// TwinCAT 3 PLC project CleanroomConnect
// ProgramVersion: 3.1.4024.0
// libraries:
//   KMWE Generic Library, * (KMWE)
//   Tc2_MC2, * (Beckhoff Automation GmbH)
//   Tc2_Standard, * (Beckhoff Automation GmbH)
//   Tc2_System, * (Beckhoff Automation GmbH)
//   Tc2_Utilities, * (Beckhoff Automation GmbH)
//   Tc3_Module, * (Beckhoff Automation GmbH)
//   VisuDialogs, * (System)
//   VisuSymbols,3.5.10.0,System
// project tree:
//   DUTs/ E_CtrlState.TcDUT (not stored), I_Door.TcIO (not stored), I_Servo.TcIO, ST_HmiBottomBar.TcDUT, ST_HmiMiddle.TcDUT, ST_HmiTopBar.TcDUT
//   / GlobalTextList.TcGTLO, MAIN.TcPOU, PlcTask.TcTTO (not stored)
//   GVLs/ GVL.TcGVL, GVL_Modules.TcGVL
//   POUs/02 UN/Unit %28UN%29/DUT/ E_AirState.TcDUT (not stored), E_ReqAction.TcDUT (not stored), E_SeqCleanroomConnect.TcDUT (not stored), ST_UN_CleanroomConnectSettings.TcDUT (not stored)
//   POUs/02 UN/Unit %28UN%29/ UN_CleanroomConnect.TcPOU (not stored)
//   POUs/03 EM/Equipment %28EM%29/2 EM_PalletConveyor/DUT/ E_ActionSelection.TcDUT (not stored), E_SeqPalletConveyor.TcDUT (not stored), I_EM_PalletConveyor.TcIO (not stored), ST_SettingsPalletConveyor.TcDUT (not stored)
//   POUs/03 EM/Equipment %28EM%29/3 EM_DockingInterface/DUTs/ I_EM_DockingInterface.TcIO (not stored), E_SeqDockingInterface.TcDUT (not stored), ST_SettingsDockingInterface.TcDUT (not stored)
//   POUs/03 EM/Equipment %28EM%29/4 EM_LiftingTransport/DUT/ E_SeqLiftingTransport.TcDUT (not stored), I_EM_LiftingTransport.TcIO (not stored), ST_PositioningProfile.TcDUT (not stored), ST_SettingsLiftingTransport.TcDUT (not stored)
//   POUs/03 EM/Equipment %28EM%29/EM_AirTreatment/DUTs/ E_SeqAirTreatment.TcDUT (not stored), I_EM_AirTreatment.TcIO (not stored), ST_SettingsAirTreatment.TcDUT (not stored)
//   POUs/03 EM/Equipment %28EM%29/EM_AirTreatment/ EM_AirTreatment.TcPOU (not stored)
//   POUs/03 EM/Equipment %28EM%29/4 EM_LiftingTransport/ EM_LiftingTransport.TcPOU (not stored)
//   POUs/03 EM/Equipment %28EM%29/1 EM_Utilities/DUTs/ E_ForceValue.TcDUT (not stored), I_EM_Utilities.TcIO (not stored), ST_SettingsUtilities.TcDUT (not stored)
//   POUs/03 EM/Equipment %28EM%29/1 EM_Utilities/ EM_Utilities.TcPOU (not stored)
//   POUs/03 EM/Equipment %28EM%29/3 EM_DockingInterface/ EM_DockingInterface.TcPOU (not stored)
//   POUs/03 EM/Equipment %28EM%29/2 EM_PalletConveyor/ EM_PalletConveyor.TcPOU (not stored)
//   POUs/04 CM/Control %28CM%29/CM_DIgitalOutput/DUT/ ST_DigOutput_HMI.TcDUT (not stored)
//   POUs/04 CM/Control %28CM%29/CM_DoorLock/DUT/ E_SeqDoorLock.TcDUT (not stored), ST_DoorLock_HMI.TcDUT (not stored), ST_SettingsDoorLock.TcDUT (not stored)
//   POUs/04 CM/Control %28CM%29/CM_MoviTrac_B/DUT/ E_SeqMoviTrac_B_WithBrake.TcDUT (not stored), I_MoviTrac_B.TcIO (not stored), ST_MoviTrac_B_HMI.TcDUT (not stored), ST_SettingsMoviTrac_B_WithBrake.TcDUT (not stored)
//   POUs/04 CM/Control %28CM%29/CM_Servo/ CM_Servo.TcPOU (not stored)
//   POUs/04 CM/Control %28CM%29/CM_Servo/DUT/ E_SeqServo.TcDUT (not stored), E_SeqInit.TcDUT (not stored), I_ServoMotor.TcIO (not stored), ST_Servo_HMI.TcDUT (not stored), ST_SettingsServo.TcDUT (not stored)
//   POUs/04 CM/Control %28CM%29/CM_DIgitalOutput/ CM_DigOutput.TcPOU (not stored)
//   POUs/04 CM/Control %28CM%29/CM_MoviTrac_B/ CM_MoviTrac_B.TcPOU (not stored)
//   POUs/04 CM/Control %28CM%29/CM_SpeedDoor/DUT/ ST_SettingsSpeedDoor.TcDUT (not stored), ST_SpeedDoor_HMI.TcDUT (not stored)
//   POUs/04 CM/Control %28CM%29/CM_TubeLedRgb/ CM_TubeLedRgb.TcPOU (not stored)
//   POUs/04 CM/Control %28CM%29/CM_TubeLedRgb/DUT/ I_LedRgb.TcIO (not stored)
//   POUs/04 CM/Control %28CM%29/CM_SpeedDoor/ CM_SpeedDoor.TcPOU (not stored)
//   POUs/04 CM/Control %28CM%29/CM_DoorLock/ CM_DoorLock.TcPOU (not stored)
//   POUs/04 CM/Control %28CM%29/CM_ValveWithFB/ CM_ValveWithDoubleFB.TcPOU (not stored), CM_ValveWithFB.TcPOU (not stored)
//   POUs/04 CM/Control %28CM%29/CM_ValveWithFB/DUT/ ST_SettingsValveWithFB.TcDUT (not stored), ST_ValveWithFB_HMI.TcDUT (not stored)
//   POUs/General/ FB_Flash.TcPOU, FB_ForceOutput.TcPOU, FB_Interlock.TcPOU (not stored), FB_InterlockHandler.TcPOU, FB_ModeStateControl.TcPOU, FB_MovAvg.TcPOU, FB_Toggle.TcPOU, F_InRange.TcPOU, ST_Interlock.TcDUT, ST_InterlockList.TcDUT, ST_MsgBox.TcDUT
// real-time tasks:
//   TASK PlcTask: cycle T#10ms, priority 20, ADS port 350
//   TASK PlcTaskHwSim: cycle T#10ms, priority 21, ADS port 351
// motion (NC):
//   TASK NC-Task 1 SAF: cycle T#2ms, priority 4, ADS port 501
//   TASK NC-Task 1 SVB: cycle T#10ms, priority 8, ADS port 511
//   AXIS TransportUnit (id 2)
//     Dynamic: AccelerationMaximum=500, DecelerationMaximum=500, Acceleration=90.006, Deceleration=90.006, Jerk=270.018
//     Velo: RefSearch=0.60004, RefSync=0.60004, SlowManual=0.5, FastManual=5, Fast=60.004, Maximum=60.004
//     PositionAreaControl: Range=0.1
//     TargetPosControl: Range=0.1
//     OtherSettings: AllowMotionCmdToSlave=true
//     encoder EncType=19
//       EncPara: ScaleFactorNumerator=180.013259, ScaleFactorDenominator=52428800, Offset=5558.46862311247, MaxCount=#xffffffff, ReferenceSystem=3
//         SoftEndMinControl: Enable=true
//         SoftEndMaxControl: Enable=true, Range=870
//         Inc: RefSearchInverse=true, RefSyncInverse=false
//     drive DrvType=16
//       DrvPara: MaxCount=#xffffffff, DriveControlDWord=#x00020100
//         Analog: VeloReferenz=66.0044, VeloScale=32, TorqueSetpointScale=10, ScaleFactorActTorque=0.1
//         TimeComp: TaskDelayCycles=1
//     controller CtrType=1
//       CtrPara: PriorControlFactor=1
//         PosDiffControl: Range=0.02
//         Observer: BandWidth=20
//   AXIS ScissorLift (id 3)
//     Dynamic: AccelerationMaximum=5, DecelerationMaximum=5, Acceleration=5, Deceleration=5, Jerk=23.436
//     Velo: RefSearch=0.05208, RefSync=0.05208, SlowManual=0.25, FastManual=2.5, Fast=5.208, Maximum=5.208
//     PositionAreaControl: Range=0.1
//     TargetPosControl: Range=0.1
//     OtherSettings: AllowMotionCmdToSlave=true, PulseDistancePos=10, PulseDistanceNeg=10
//     encoder EncType=8
//       EncPara: ScaleFactorNumerator=6, ScaleFactorDenominator=50331648, Offset=46.5910750851166, MaxCount=#xffffffff, ReferenceSystem=3
//         SoftEndMinControl: Enable=true
//         SoftEndMaxControl: Enable=true, Range=152
//         Inc: RefSearchInverse=true, RefSyncInverse=false
//     drive DrvType=9
//       DrvPara: MaxCount=#xffffffff, DriveControlDWord=#x00030100
//         Analog: VeloReferenz=5.7288, VeloScale=1.02400649589962, TorqueSetpointScale=10, ScaleFactorActTorque=0.1
//         TimeComp: TaskDelayCycles=1
//     controller CtrType=1
//       CtrPara: PriorControlFactor=1
//         PosDiffControl: Range=0.01
//         Observer: BandWidth=20
// I/O:
//   DEVICE Master (EtherCAT), AmsNetId 5.152.40.20.4.1
//     K1 (EK1200) [EK1200-5000 EtherCAT Power supply (2A E-Bus)]
//       K2 (EL6070-0033) [EL6070-0033 1Ch. Licence key terminal, individual licences]
//       K3 (EL1809) [EL1809 16Ch. Dig. Input 24V, 3ms]
//       K4 (EL1809) [EL1809 16Ch. Dig. Input 24V, 3ms]
//       K5 (EL1809) [EL1809 16Ch. Dig. Input 24V, 3ms]
//       K6 (EL1809) [EL1809 16Ch. Dig. Input 24V, 3ms]
//       K7 (EL2809) [EL2809 16Ch. Dig. Output 24V, 0.5A]
//       K8 (EL4024) [EL4024 4Ch. Ana. Output 4-20mA, 12bit]
//       K9 (EL7211-9014) [EL7211-9014 1Ch. MDP742 Servo motor output stage with OCT (50V, 4.5A RMS) and STO input]
//         startup 32785:21 := 0E01 // DRV Motor Settings / Commutation offset
//         startup 32786:19 := 0000 // DRV Brake Settings / Emergency application timeout
//         startup 32784:51 := 0A00 // DRV Amplifier Settings / Stand still window
//         startup 32785:27 := 4F080000 // DRV Motor Settings / Motor speed limitation
//         startup 28688:3 := 09 // DRV Outputs / Modes of operation
//         startup 32784:87 := 64 // DRV Amplifier Settings / Velocity feed forward gain
//         startup 28688:11 := D007 // DRV Outputs / Torque limitation
//         startup 32784:19 := 8701 // DRV Amplifier Settings / Current loop proportional gain
//         startup 32784:18 := 0500 // DRV Amplifier Settings / Current loop integral time
//         startup 32784:21 := 92000000 // DRV Amplifier Settings / Velocity loop proportional gain
//         startup 32784:20 := 96000000 // DRV Amplifier Settings / Velocity loop integral time
//         startup 32768:1 := 00 // FB Settings / Invert feedback direction
//       K10 (EL9576) [EL9576 Brake chopper terminal]
//       K11 (EL2904) [EL2904, 4 Ch. Safety Output 24V, 0.5A, TwinSAFE]
//         modules: Module 1 (FSOES), Module 2 (DO)
//       K12 (EL1918 + TwinSAFE Logic)
//       K20 (EL9110) [EL9110 Power Supplier with LED (24V, Diagnostics)]
//       K21 (EL2809) [EL2809 16Ch. Dig. Output 24V, 0.5A]
//       K22 (EL9011) [EL9011 End Terminal]
//   DEVICE Master Field (EtherCAT), AmsNetId 5.152.40.20.5.1
//     U9 (AX5103-0000-0215) [AX5103-0000-0215 EtherCAT Drive (SoE, 1 Ch.)]
//       Term 3 (AX5805) [AX5805 (Safety Drive Option)]
//         modules: Module 1 (Safety Process Data, 1 axis), Module 2 (Standard Process Data, 1 axis)
//       Term 3 (EL9011) [EL9011 End Terminal]
// variable links:
//   Master (EtherCAT) <-> Master (EtherCAT)/K1 (EK1200)/K12 (EL1918 + TwinSAFE Logic)
//     K1 (EK1200)/K11 (EL2904)/Module 1 (FSOES)/RxPDO/FSOE <-> ConnectionInputs/TwinSafeGroup1.EL2904, 4 digital outputs_1_22 TxPDO
//     K1 (EK1200)/K11 (EL2904)/Module 1 (FSOES)/TxPDO/FSOE <-> ConnectionOutputs/TwinSafeGroup1.EL2904, 4 digital outputs_1_22 RxPDO
//   Master (EtherCAT) <-> Master Field (EtherCAT)/U9 (AX5103-0000-0215)/Term 3 (AX5805)
//     K1 (EK1200)/K12 (EL1918 + TwinSAFE Logic)/ConnectionInputs/TwinSafeGroup1.AX5805, Safety Process Data 1 axis_37 TxPDO <-> Module 1 (Safety Process Data, 1 axis)/Outputs (Controlword)/FSOE
//     K1 (EK1200)/K12 (EL1918 + TwinSAFE Logic)/ConnectionOutputs/TwinSafeGroup1.AX5805, Safety Process Data 1 axis_37 RxPDO <-> Module 1 (Safety Process Data, 1 axis)/Inputs (Statusword)/FSOE
//   NC-Task 1 SAF/Axes/TransportUnit <-> Master (EtherCAT)/K1 (EK1200)/K9 (EL7211-9014)
//     Drive/Inputs/In/nDataIn1 <-> DRV Following error actual value/Following error actual value
//     Drive/Inputs/In/nDataIn3[0] <-> DRV Torque actual value/Torque actual value
//     Drive/Inputs/In/nDcOutputTime <-> InfoData/DcOutputShift
//     Drive/Inputs/In/nState1 <-> DRV Statusword/Statusword
//     Drive/Inputs/In/nState2 <-> DRV Statusword/Statusword @bit 8
//     Drive/Inputs/In/nState4 @bit 1 <-> WcState/InputToggle
//     Drive/Inputs/In/nState4 <-> WcState/WcState
//     Drive/Outputs/Out/nCtrl1 <-> DRV Controlword/Controlword
//     Drive/Outputs/Out/nCtrl2 <-> DRV Controlword/Controlword @bit 8
//     Drive/Outputs/Out/nDataOut1 <-> DRV Target position/Target position
//     Drive/Outputs/Out/nDataOut2 <-> DRV Target velocity/Target velocity
//     Enc/Inputs/In/nDataIn1 <-> FB Position/Position
//     Enc/Inputs/In/nDcInputTime <-> InfoData/DcInputShift
//     Enc/Inputs/In/nState4 @bit 1 <-> WcState/InputToggle
//     Enc/Inputs/In/nState4 <-> WcState/WcState
//   CleanroomConnect/CleanroomConnect Instance <-> Master (EtherCAT)/K1 (EK1200)/K10 (EL9576)
//     PlcTask Inputs/GVL_Modules.g_emLiftingTransport.I_bErrI2Terror <-> BCT Inputs/I2T error
//     PlcTask Inputs/GVL_Modules.g_emLiftingTransport.I_bErrOvervoltage <-> BCT Inputs/Overvoltage
//     PlcTask Inputs/GVL_Modules.g_emLiftingTransport.I_bErrTerminalOvertemperature <-> BCT Inputs/Terminal Overtemperature
//     PlcTask Inputs/GVL_Modules.g_emLiftingTransport.I_berrOvercurrentProtection <-> BCT Inputs/Overcurrent Protection
//     PlcTask Inputs/GVL_Modules.g_emLiftingTransport.I_bwrnI2Twarning <-> BCT Inputs/I2T warning
//     PlcTask Inputs/GVL_Modules.g_emLiftingTransport.I_bwrnUndervoltage <-> BCT Inputs/Undervoltage
//   CleanroomConnect/CleanroomConnect Instance <-> Master (EtherCAT)/K1 (EK1200)/K12 (EL1918 + TwinSAFE Logic)
//     PlcTask Inputs/GVL_Modules.g_emLiftingTransport.s_cmLift.I_bEnable <-> StandardInputs/TwinSafeGroup1.ScissorLift_EnableNC_26
//     PlcTask Inputs/GVL_Modules.g_emLiftingTransport.s_cmTransport.I_bEnable <-> StandardInputs/TwinSafeGroup1.TransportUnit_EnableNC_27
//     PlcTask Inputs/GVL_Modules.g_emUtilities.I_nStaInputSafeDataByte0 <-> Device Info Data/Internal I/O/Input Safe Data Byte 0
//     PlcTask Inputs/GVL_Modules.g_emUtilities.I_nStaInputSafeDataByte1 <-> Device Info Data/Internal I/O/Input Safe Data Byte 1
//     PlcTask Inputs/GVL_Modules.g_emUtilities.I_nTwinSATE_ProjectCrc <-> Device Info Data/Project CRC
//     PlcTask Inputs/GVL_Modules.g_emUtilities.s_diSafetyFbErr.I_bStaInput <-> StandardInputs/TwinSafeGroup1.FB_Err_24
//     PlcTask Inputs/GVL_Modules.g_emUtilities.s_diSafetyOk.I_bStaInput <-> StandardInputs/TwinSafeGroup1.SafetyOK_29
//     PlcTask Outputs/GVL_Modules.g_emLiftingTransport.Q_bDriveStateSTO <-> StandardOutputs/TwinSafeGroup1.FbTransportUnit_STO_28
//     PlcTask Outputs/GVL_Modules.g_emUtilities.Q_bCmdErrAck <-> StandardOutputs/TwinSafeGroup1.ErrorAcknowledgement_1
//     PlcTask Outputs/GVL_Modules.g_emUtilities.Q_bCmdRestartSafety <-> StandardOutputs/TwinSafeGroup1.RestartSafety_5
//     PlcTask Outputs/GVL_Modules.g_emUtilities.Q_bCmdRun <-> StandardOutputs/TwinSafeGroup1.Run_2
//   CleanroomConnect/CleanroomConnect Instance <-> Master (EtherCAT)/K1 (EK1200)/K20 (EL9110)
//     PlcTask Inputs/GVL_Modules.g_emUtilities.s_diPowerPotentialGroup24VdcOk.I_bStaInput <-> PowerOK/Input
//   CleanroomConnect/CleanroomConnect Instance <-> Master (EtherCAT)/K1 (EK1200)/K21 (EL2809)
//     PlcTask Outputs/GVL_Modules.g_emDockingInterface.s_cmClampsLowerHighPressure.Q_bStaOutput <-> Channel 8/Output
//     PlcTask Outputs/GVL_Modules.g_emDockingInterface.s_cmClampsUpperHighPressure.Q_bStaOutput <-> Channel 7/Output
//     PlcTask Outputs/GVL_Modules.g_emDockingInterface.s_cmDockingClampsLower.Q_bCmdOff <-> Channel 6/Output
//     PlcTask Outputs/GVL_Modules.g_emDockingInterface.s_cmDockingClampsLower.Q_bCmdOn <-> Channel 5/Output
//     PlcTask Outputs/GVL_Modules.g_emDockingInterface.s_cmDockingClampsUpper.Q_bCmdOff <-> Channel 4/Output
//     PlcTask Outputs/GVL_Modules.g_emDockingInterface.s_cmDockingClampsUpper.Q_bCmdOn <-> Channel 3/Output
//     PlcTask Outputs/GVL_Modules.g_emDockingInterface.s_cmDoorOpener.Q_bCmdOff <-> Channel 14/Output
//     PlcTask Outputs/GVL_Modules.g_emDockingInterface.s_cmDoorOpener.Q_bCmdOn <-> Channel 13/Output
//     PlcTask Outputs/GVL_Modules.g_emDockingInterface.s_cmDoorShutter.Q_bCmdOff <-> Channel 16/Output
//     PlcTask Outputs/GVL_Modules.g_emDockingInterface.s_cmDoorShutter.Q_bCmdOn <-> Channel 15/Output
//     PlcTask Outputs/GVL_Modules.g_emDockingInterface.s_cmUnlockingPinLower.Q_bCmdOff <-> Channel 12/Output
//     PlcTask Outputs/GVL_Modules.g_emDockingInterface.s_cmUnlockingPinLower.Q_bCmdOn <-> Channel 11/Output
//     PlcTask Outputs/GVL_Modules.g_emDockingInterface.s_cmUnlockingPinUpper.Q_bCmdOff <-> Channel 10/Output
//     PlcTask Outputs/GVL_Modules.g_emDockingInterface.s_cmUnlockingPinUpper.Q_bCmdOn <-> Channel 9/Output
//     PlcTask Outputs/GVL_Modules.g_emPalletConveyor.s_cmCenteringUnit.Q_bCmdOff <-> Channel 2/Output
//     PlcTask Outputs/GVL_Modules.g_emPalletConveyor.s_cmCenteringUnit.Q_bCmdOn <-> Channel 1/Output
//   CleanroomConnect/CleanroomConnect Instance <-> Master (EtherCAT)/K1 (EK1200)/K3 (EL1809)
//     PlcTask Inputs/GVL_Modules.g_emUtilities.s_diAirPressureOk.I_bStaInput <-> Channel 7/Input
//     PlcTask Inputs/GVL_Modules.g_emUtilities.s_diCabinetTemperatureOk.I_bStaInput <-> Channel 8/Input
//     PlcTask Inputs/GVL_Modules.g_emUtilities.s_diPower230VacOk.I_bStaInput <-> Channel 3/Input
//     PlcTask Inputs/GVL_Modules.g_emUtilities.s_diPower400VacOk.I_bStaInput <-> Channel 2/Input
//     PlcTask Inputs/GVL_Modules.g_emUtilities.s_diPower230VacSocketsOk.I_bStaInput <-> Channel 4/Input
//     PlcTask Inputs/GVL_Modules.g_emUtilities.s_diPower48VdcOk.I_bStaInput <-> Channel 5/Input
//     PlcTask Inputs/GVL_Modules.g_emUtilities.s_diRestartSafety.I_bStaInput <-> Channel 1/Input
//   CleanroomConnect/CleanroomConnect Instance <-> Master (EtherCAT)/K1 (EK1200)/K4 (EL1809)
//     PlcTask Inputs/GVL_Modules.g_emDockingInterface.s_cmDockingClampsLower.I_bStaValveIsOff <-> Channel 16/Input
//     PlcTask Inputs/GVL_Modules.g_emDockingInterface.s_cmDockingClampsUpper.I_bStaValveIsOff <-> Channel 12/Input
//     PlcTask Inputs/GVL_Modules.g_emDockingInterface.s_cmDockingClampsUpper.I_bStaValveIsOff2 <-> Channel 14/Input
//     PlcTask Inputs/GVL_Modules.g_emDockingInterface.s_cmDockingClampsUpper.I_bStaValveIsOn <-> Channel 13/Input
//     PlcTask Inputs/GVL_Modules.g_emDockingInterface.s_cmDockingClampsUpper.I_bStaValveIsOn2 <-> Channel 15/Input
//     PlcTask Inputs/GVL_Modules.g_emPalletConveyor.s_cmCenteringUnit.I_bStaValveIsOff <-> Channel 8/Input
//     PlcTask Inputs/GVL_Modules.g_emPalletConveyor.s_cmCenteringUnit.I_bStaValveIsOff2 <-> Channel 10/Input
//     PlcTask Inputs/GVL_Modules.g_emPalletConveyor.s_cmCenteringUnit.I_bStaValveIsOn <-> Channel 9/Input
//     PlcTask Inputs/GVL_Modules.g_emPalletConveyor.s_cmCenteringUnit.I_bStaValveIsOn2 <-> Channel 11/Input
//     PlcTask Inputs/GVL_Modules.g_emPalletConveyor.s_cmPalletConveyor.I_bStaMotorIsRunning <-> Channel 7/Input
//     PlcTask Inputs/GVL_Modules.g_emPalletConveyor.s_cmPalletConveyor.I_bStaReadyForOperation <-> Channel 6/Input
//     PlcTask Inputs/GVL_Modules.g_emPalletConveyor.s_diStaAtCenteringPosition.I_bStaInput <-> Channel 3/Input
//     PlcTask Inputs/GVL_Modules.g_emPalletConveyor.s_diStaAtDockingPosition.I_bStaInput <-> Channel 4/Input
//     PlcTask Inputs/GVL_Modules.g_emPalletConveyor.s_diStaAtInfeedPositionFront.I_bStaInput <-> Channel 2/Input
//     PlcTask Inputs/GVL_Modules.g_emPalletConveyor.s_diStaAtInfeedPositionRear.I_bStaInput <-> Channel 1/Input
//     PlcTask Inputs/GVL_Modules.g_emPalletConveyor.s_diStaDoorOpened.I_bStaInput <-> Channel 5/Input
//   CleanroomConnect/CleanroomConnect Instance <-> Master (EtherCAT)/K1 (EK1200)/K5 (EL1809)
//     PlcTask Inputs/GVL_Modules.g_emDockingInterface.s_cmDockingClampsLower.I_bStaValveIsOff2 <-> Channel 2/Input
//     PlcTask Inputs/GVL_Modules.g_emDockingInterface.s_cmDockingClampsLower.I_bStaValveIsOn <-> Channel 1/Input
//     PlcTask Inputs/GVL_Modules.g_emDockingInterface.s_cmDockingClampsLower.I_bStaValveIsOn2 <-> Channel 3/Input
//     PlcTask Inputs/GVL_Modules.g_emDockingInterface.s_cmDoorOpener.I_bStaValveIsOff <-> Channel 8/Input
//     PlcTask Inputs/GVL_Modules.g_emDockingInterface.s_cmDoorOpener.I_bStaValveIsOn <-> Channel 9/Input
//     PlcTask Inputs/GVL_Modules.g_emDockingInterface.s_cmDoorShutter.I_bStaValveIsOff <-> Channel 11/Input
//     PlcTask Inputs/GVL_Modules.g_emDockingInterface.s_cmDoorShutter.I_bStaValveIsOn <-> Channel 12/Input
//     PlcTask Inputs/GVL_Modules.g_emDockingInterface.s_cmUnlockingPinLower.I_bStaValveIsOff <-> Channel 6/Input
//     PlcTask Inputs/GVL_Modules.g_emDockingInterface.s_cmUnlockingPinLower.I_bStaValveIsOn <-> Channel 7/Input
//     PlcTask Inputs/GVL_Modules.g_emDockingInterface.s_cmUnlockingPinUpper.I_bStaValveIsOff <-> Channel 4/Input
//     PlcTask Inputs/GVL_Modules.g_emDockingInterface.s_cmUnlockingPinUpper.I_bStaValveIsOn <-> Channel 5/Input
//     PlcTask Inputs/GVL_Modules.g_emDockingInterface.s_diStaDoorAlmostClosed.I_bStaInput <-> Channel 10/Input
//   CleanroomConnect/CleanroomConnect Instance <-> Master (EtherCAT)/K1 (EK1200)/K6 (EL1809)
//     PlcTask Inputs/GVL_Modules.g_emLiftingTransport.s_cmLift.I_bDetLimitSwitchNeg <-> Channel 1/Input
//     PlcTask Inputs/GVL_Modules.g_emLiftingTransport.s_cmLift.I_bDetLimitSwitchPos <-> Channel 2/Input
//     PlcTask Inputs/GVL_Modules.g_emLiftingTransport.s_cmLift.I_bDetReferenceSwitch <-> Channel 3/Input
//     PlcTask Inputs/GVL_Modules.g_emLiftingTransport.s_cmTransport.I_bDetLimitSwitchNeg <-> Channel 9/Input
//     PlcTask Inputs/GVL_Modules.g_emLiftingTransport.s_cmTransport.I_bDetLimitSwitchPos <-> Channel 10/Input
//     PlcTask Inputs/GVL_Modules.g_emLiftingTransport.s_cmTransport.I_bDetReferenceSwitch <-> Channel 11/Input
//     PlcTask Inputs/GVL_Modules.g_emLiftingTransport.s_diStaCabinAreaOccupied.I_bStaInput <-> Channel 12/Input
//     PlcTask Inputs/GVL_Modules.g_emLiftingTransport.s_diStaCollisionAvoidanceSensor.I_bStaInput <-> Channel 6/Input
//     PlcTask Inputs/GVL_Modules.g_emLiftingTransport.s_diStaTrolleyLocked.I_bStaInput <-> Channel 13/Input
//     PlcTask Inputs/GVL_Modules.g_emLiftingTransport.s_diStaTrolleyOnPositionLeft.I_bStaInput <-> Channel 4/Input
//     PlcTask Inputs/GVL_Modules.g_emLiftingTransport.s_diStaTrolleyOnPositionRight.I_bStaInput <-> Channel 5/Input
//   CleanroomConnect/CleanroomConnect Instance <-> Master (EtherCAT)/K1 (EK1200)/K7 (EL2809)
//     PlcTask Outputs/GVL_Modules.g_emPalletConveyor.s_cmPalletConveyor.Q_bCmdEnable <-> Channel 6/Output
//     PlcTask Outputs/GVL_Modules.g_emPalletConveyor.s_cmPalletConveyor.Q_bCmdReleaseBrake <-> Channel 9/Output
//     PlcTask Outputs/GVL_Modules.g_emPalletConveyor.s_cmPalletConveyor.Q_bCmdReset <-> Channel 5/Output
//     PlcTask Outputs/GVL_Modules.g_emPalletConveyor.s_cmPalletConveyor.Q_bCmdStartCCW <-> Channel 8/Output
//     PlcTask Outputs/GVL_Modules.g_emPalletConveyor.s_cmPalletConveyor.Q_bCmdStartCW <-> Channel 7/Output
//     PlcTask Outputs/GVL_Modules.g_emUtilities.s_doBeaconLedGreen.Q_bStaOutput <-> Channel 3/Output
//     PlcTask Outputs/GVL_Modules.g_emUtilities.s_doBeaconLedRed.Q_bStaOutput <-> Channel 1/Output
//     PlcTask Outputs/GVL_Modules.g_emUtilities.s_doBeaconLedYellow.Q_bStaOutput <-> Channel 2/Output
//     PlcTask Outputs/GVL_Modules.g_emUtilities.s_doSnRestartSafety.Q_bStaOutput <-> Channel 10/Output
//   CleanroomConnect/CleanroomConnect Instance <-> Master (EtherCAT)/K1 (EK1200)/K8 (EL4024)
//     PlcTask Outputs/GVL_Modules.g_emPalletConveyor.s_cmPalletConveyor.Q_nSetTargetSpeed <-> AO Outputs Channel 1/Analog output
//   CleanroomConnect/CleanroomConnect Instance <-> Master (EtherCAT)/K1 (EK1200)/K9 (EL7211-9014)
//     PlcTask Inputs/GVL_Modules.g_emLiftingTransport.I_nInfoDataInputLevel <-> DRV Info data 1/Info data 1
//   CleanroomConnect/CleanroomConnect Instance <-> NC-Task 1 SAF/Axes/ScissorLift
//     PlcTask Inputs/GVL_Modules.g_emLiftingTransport.axisLift.NcToPlc <-> Outputs/ToPlc
//     PlcTask Outputs/GVL_Modules.g_emLiftingTransport.axisLift.PlcToNc <-> Inputs/FromPlc
//   CleanroomConnect/CleanroomConnect Instance <-> NC-Task 1 SAF/Axes/TransportUnit
//     PlcTask Inputs/GVL_Modules.g_emLiftingTransport.axisTransport.NcToPlc <-> Outputs/ToPlc
//     PlcTask Outputs/GVL_Modules.g_emLiftingTransport.axisTransport.PlcToNc <-> Inputs/FromPlc
//   (this object) <-> Master Field (EtherCAT)/U9 (AX5103-0000-0215)
//     Drive/Inputs/In/nDataIn1 <-> AT/Following distance
//     Drive/Inputs/In/nDataIn3[0] <-> AT/Torque/force feedback value
//     Drive/Inputs/In/nDcOutputTime <-> InfoData/DcOutputShift
//     Drive/Inputs/In/nState1 <-> AT/Drive status word @bit 8
//     Drive/Inputs/In/nState2 <-> AT/Drive status word
//     Drive/Inputs/In/nState4 @bit 1 <-> WcState/InputToggle
//     Drive/Inputs/In/nState4 <-> WcState/WcState
//     Drive/Outputs/Out/nCtrl1 <-> MDT/Master control word @bit 8
//     Drive/Outputs/Out/nDataOut1 <-> MDT/Position command value
//     Enc/Inputs/In/nDataIn1 <-> AT/Position feedback 1 value
//     Enc/Inputs/In/nDcInputTime <-> InfoData/DcInputShift
//     Enc/Inputs/In/nState4 @bit 1 <-> WcState/InputToggle
//     Enc/Inputs/In/nState4 <-> WcState/WcState

// ---- DUTs/ST_HmiBottomBar.TcDUT
TYPE ST_HmiBottomBar :
STRUCT CONSTANT
	Start					: STRING := 'WebContent/Bottom/NavigationBarStart.content';
	Alarm					: STRING := 'WebContent/Bottom/NavigationBarAlarm.content';
	General_ReturnToStart	: STRING := 'WebContent/Bottom/NavigationBarReturnToStart.content';
END_STRUCT
END_TYPE

// ---- DUTs/ST_HmiMiddle.TcDUT
TYPE ST_HmiMiddle :
STRUCT CONSTANT 
	//General Pages
	Start 				: STRING := 'WebContent/Middle/Start.content';
	AlarmManager 		: STRING := 'WebContent/Middle/AlarmManager.content';
	ParameterManager 	: STRING := 'WebContent/Middle/ParameterManager.content';
	
	//Units
	UN_CleanroomConnect	: STRING := 'WebContent/Middle/UN_CleanroomConnect/UN_CleanroomConnect.content';
	
	//Equipment Modules
	EM_Utilities		: STRING := 'WebContent/Middle/EM_Utilities/EM_Utilities.content';
	EM_PalletConveyor	: STRING := 'WebContent/Middle/EM_PalletConveyor/EM_PalletConveyor.content';
	EM_DockingInterface	: STRING := 'WebContent/Middle/EM_DockingInterface/EM_DockingInterface.content';
	EM_LiftingTransport	: STRING := 'WebContent/Middle/EM_LiftingTransport/EM_LiftingTransport.content';
//++EM_AirTreatment		: STRING := 'WebContent/Middle/EM_AirTreatment/EM_AirTreatment.content';

END_STRUCT
END_TYPE

// ---- DUTs/ST_HmiTopBar.TcDUT
TYPE ST_HmiTopBar :
STRUCT CONSTANT 
	GeneralTopbar : STRING := 'WebContent/Top/TopBar.content';
END_STRUCT
END_TYPE

// ---- POUs/General/ST_Interlock.TcDUT
TYPE ST_Interlock :
STRUCT
	bState : BOOL := FALSE;
	sReason : STRING(GVL.g_nMAX_LEN_REASON) := 'none';
END_STRUCT
END_TYPE

// ---- POUs/General/ST_InterlockList.TcDUT
TYPE ST_InterlockList :
STRUCT
	arr_Interlocks : ARRAY[0..GVL.g_nLEN_INTERLOCK_LIST-1] OF ST_Interlock;
END_STRUCT
END_TYPE

// ---- POUs/General/ST_MsgBox.TcDUT
TYPE ST_MsgBox :
STRUCT
	bShow : BOOL := FALSE;
	bBtnPressed : BOOL := FALSE;
	sMessageText : STRING(64) := '_just_a_message_';
	sResponse : STRING(32) := '_just_an_response_';
END_STRUCT
END_TYPE

// ---- GVLs/GVL.TcGVL
{attribute 'qualified_only'}
VAR_GLOBAL
	g_unCleanroomConnect : UN_CleanroomConnect;
	
	g_bLedFlashSlow : BOOL;
	g_bLedFlashFast : BOOL;
	
	g_sUser : STRING;
	g_sSerialNumber : STRING;
	g_sNotesEntry : T_MAXSTRING;
	
	//Hmi linked variable
	g_sToHmiTopContent : STRING;
	g_sToHmiMiddleContent : STRING;
	g_sToHmiMiddleTab : STRING;
	g_sToHmiBottomContent : STRING;
	
	//Structs with screens that can be appointed to linked variables
	g_stHmiTopBar : ST_HmiTopBar;
	g_stHmiMiddle : ST_HmiMiddle;
	g_stHmiBottomBar : ST_HmiBottomBar;
	
	g_osrNotify : R_TRIG;
END_VAR

VAR_GLOBAL CONSTANT
	g_nMAX_LEN_FEEDBACK : USINT := 8; //Used in CM's
	g_nMAX_LEN_STEP_NAME : USINT := 32;
	g_nMAX_LEN_REASON : USINT := 96;
	g_nLEN_INTERLOCK_LIST : USINT := 6;
	
	g_bFUMO3_Enabled : BOOL := FALSE;
END_VAR

// ---- GVLs/GVL_Modules.TcGVL
{attribute 'qualified_only'}
VAR_GLOBAL
	g_emUtilities : EM_Utilities;
	g_emPalletConveyor : EM_PalletConveyor;
	g_emDockingInterface : EM_DockingInterface;
	g_emLiftingTransport : EM_LiftingTransport;
	g_emAirTreatment : EM_AirTreatment;
END_VAR

// ---- DUTs/I_Servo.TcIO
INTERFACE I_Servo

METHOD PUBLIC m_MC_Home : BOOL
VAR_INPUT
	i_bExecute : BOOL;
	i_fPosition : REAL;
	i_eHomingMode : TC2_MC2.MC_HomingMode;
	i_eBufferMode : TC2_MC2.MC_BufferMode;
END_VAR
END_METHOD

METHOD PUBLIC m_MC_Jog : BOOL
VAR_INPUT
	i_bExecute : BOOL;
	i_bJogForward : BOOL;
	i_bJogBackward : BOOL;
	i_eJogMode : TC2_MC2.E_JogMode;
	i_fPosition : LREAL; 
	i_fVelocity : LREAL; 
	i_fAcceleration : LREAL; 
	i_fDeceleration : LREAL; 
	i_fJerk : LREAL;
END_VAR
END_METHOD

METHOD PUBLIC m_MC_MoveAbsolute : BOOL
VAR_INPUT
	i_bExecute : BOOL;
	i_fPosition : LREAL; 
	i_fVelocity : LREAL; 
	i_fAcceleration : LREAL; 
	i_fDeceleration : LREAL; 
	i_fJerk : LREAL;
	i_eBufferMode : TC2_MC2.MC_BufferMode;
END_VAR

VAR_OUTPUT
	o_Busy : BOOL;
	o_bDone : BOOL;
	o_bError : BOOL;
END_VAR
END_METHOD

METHOD PUBLIC m_MC_MoveRelative : BOOL
VAR_INPUT
	i_bExecute : BOOL;
	i_fDistance : LREAL; 
	i_fVelocity : LREAL; 
	i_fAcceleration : LREAL; 
	i_fDeceleration : LREAL; 
	i_fJerk : LREAL;
	i_eBufferMode : TC2_MC2.MC_BufferMode;
END_VAR
END_METHOD

METHOD PUBLIC m_MC_MoveVelocity : BOOL
VAR_INPUT
	i_bExecute : BOOL;
	i_fVelocity : LREAL; 
	i_fAcceleration : LREAL; 
	i_fDeceleration : LREAL; 
	i_fJerk : LREAL;
	i_eDirection : TC2_MC2.MC_Direction;
	i_eBufferMode : TC2_MC2.MC_BufferMode;
END_VAR
END_METHOD

METHOD PUBLIC m_MC_Power : BOOL
VAR_INPUT
	i_bEnable : BOOL;
	i_bEnablePositive : BOOL;
	i_bEnableNegative : BOOL;
	i_fOverride : LREAL;
	i_eBufferMode : TC2_MC2.MC_BufferMode;
END_VAR
END_METHOD

METHOD PUBLIC m_MC_Reset : BOOL
VAR_INPUT
	i_bExecute : BOOL;
END_VAR
END_METHOD

METHOD PUBLIC m_MC_Stop : BOOL
VAR_INPUT
	i_bExecute : BOOL;
	i_fDeceleration : LREAL;
	i_fJerk : LREAL;
END_VAR
END_METHOD

PROPERTY PUBLIC p_bActive : BOOL
GET
END_GET
END_PROPERTY

PROPERTY PUBLIC p_bAtPosition : BOOL
GET
END_GET
END_PROPERTY

PROPERTY PUBLIC p_bBusy : BOOL
GET
END_GET
END_PROPERTY

PROPERTY PUBLIC p_bCommandAborted : BOOL
GET
END_GET
END_PROPERTY

PROPERTY PUBLIC p_bDone : BOOL
GET
END_GET
END_PROPERTY

PROPERTY PUBLIC p_bError : BOOL
GET
END_GET
END_PROPERTY

PROPERTY PUBLIC p_bHomed : BOOL
GET
END_GET
END_PROPERTY

PROPERTY PUBLIC p_bInVelocity : BOOL
GET
END_GET
END_PROPERTY

PROPERTY PUBLIC p_bStandstill : BOOL
GET
END_GET
END_PROPERTY

PROPERTY PUBLIC p_fPosition : LREAL
GET
END_GET
END_PROPERTY

PROPERTY PUBLIC p_fVelocity : LREAL
GET
END_GET
END_PROPERTY

PROPERTY PUBLIC p_nErrorID : UDINT
GET
END_GET
END_PROPERTY

END_INTERFACE

// ---- MAIN.TcPOU
PROGRAM MAIN
VAR
	s_ParamPathnames : ARRAY[1..Param_Project.n_MaxParamFolders] OF STRING := ['C:\Cleanroom_Connect\Parameters'];
	
	User : STRING := '<user_name>';
	SoftwareVersion : STRING := '<software_version>';
	InitDone : BOOL;
	Shutdown : BOOL;
	
	fbModeStateControl : FB_ModeStateControl;
END_VAR

GVL_KMWEGenericLib.g_fbAlarmManager();

GVL_KMWEGenericLib.g_fbParamManager.p_bShowHmiParam := TRUE;

GVL_KMWEGenericLib.g_fbParamManager(
	i_sPathName := s_ParamPathnames,
	i_osrResetImportExport := GVL_KMWEGenericLib.g_fbAlarmManager.p_osrReset);

fbModeStateControl();

GVL.g_unCleanroomConnect.p_bCmdReset := GVL_KMWEGenericLib.g_fbAlarmManager.p_osrReset;
GVL.g_unCleanroomConnect();

END_PROGRAM

// ---- POUs/General/FB_ModeStateControl.TcPOU
FUNCTION_BLOCK FB_ModeStateControl
VAR_INPUT
	i_bReqStopAlarm	: BOOL;
	i_bStaAllStopped : BOOL;
END_VAR
VAR
	s_bInitDone : BOOL := FALSE;
	
	s_eCtrlMode : E_CtrlMode := E_CtrlMode.IDLE;
	s_eCtrlState : E_CtrlState := E_CtrlState.STOPPED;
	
	s_fbHmiBtnModeAutomatic : FB_HmiBtn;
	s_fbHmiBtnModeManual : FB_HmiBtn;
	s_fbHmiBtnModeMaintenance : FB_HmiBtn;
	s_fbHmiBtnModeIO : FB_HmiBtn;
	s_fbHmiBtnModeCleaning : FB_HmiBtn;
	
	s_fbHmiBtnStateStart : FB_HmiBtn;
	s_fbHmiBtnStateStop : FB_HmiBtn;
	s_fbHmiBtnStateReset : FB_HmiBtn;
END_VAR


m_Main();

METHOD PROTECTED _m_Devices : BOOL

//Mode buttons
s_fbHmiBtnModeAutomatic();
s_fbHmiBtnModeManual();
s_fbHmiBtnModeMaintenance();
s_fbHmiBtnModeIO();
s_fbHmiBtnModeCleaning();

//State buttons
s_fbHmiBtnStateStart();
s_fbHmiBtnStateStop();
s_fbHmiBtnStateReset();

CASE s_eCtrlMode OF
	E_CtrlMode.IDLE:
		s_fbHmiBtnModeAutomatic.p_bStaVisible := TRUE;
		s_fbHmiBtnModeManual.p_bStaVisible := TRUE;
		s_fbHmiBtnModeMaintenance.p_bStaVisible := TRUE;
		s_fbHmiBtnModeIO.p_bStaVisible := TRUE;
		s_fbHmiBtnModeCleaning.p_bStaVisible := TRUE;
		
		s_fbHmiBtnStateStart.p_bStaVisible := TRUE;
		s_fbHmiBtnStateStop.p_bStaVisible := TRUE;
		s_fbHmiBtnStateReset.p_bStaVisible := TRUE;
		
	E_CtrlMode.AUTOMATIC:
		;
		
	E_CtrlMode.MANUAL:
		;
		
	E_CtrlMode.MAINTENANCE:
		;
		
	E_CtrlMode.IO:
		;
		
	E_CtrlMode.CLEANING:
		;
	ELSE
		s_eCtrlMode := E_CtrlMode.IDLE;
END_CASE

IF (s_eCtrlState = E_CtrlState.STOPPED) THEN
		IF s_fbHmiBtnModeAutomatic.p_osrBtnPress THEN
			s_eCtrlMode := E_CtrlMode.AUTOMATIC;
			
		ELSIF s_fbHmiBtnModeManual.p_osrBtnPress THEN
			s_eCtrlMode := E_CtrlMode.MANUAL;
			
		ELSIF s_fbHmiBtnModeMaintenance.p_osrBtnPress THEN
			s_eCtrlMode := E_CtrlMode.MAINTENANCE;
			
		ELSIF s_fbHmiBtnModeIO.p_osrBtnPress THEN
			s_eCtrlMode := E_CtrlMode.IO;
			
		ELSIF s_fbHmiBtnModeCleaning.p_osrBtnPress THEN
			s_eCtrlMode := E_CtrlMode.CLEANING;
			
		END_IF
	END_IF

CASE s_eCtrlState OF
	E_CtrlState.STOPPED:
		
		IF s_fbHmiBtnStateReset.p_osrBtnPress THEN
			s_eCtrlState := E_CtrlState.IDLE;
		END_IF 
		
	E_CtrlState.IDLE:
		
		IF s_fbHmiBtnStateStop.p_osrBtnPress THEN
			s_eCtrlState := E_CtrlState.STOPPING;
		ELSIF s_fbHmiBtnStateStart.p_osrBtnPress THEN
			s_eCtrlState := E_CtrlState.RUNNING;
		END_IF
		
	E_CtrlState.RUNNING:
		
		IF s_fbHmiBtnStateStop.p_osrBtnPress OR i_bReqStopAlarm THEN
			s_eCtrlState := E_CtrlState.STOPPING;
		END_IF
		
	E_CtrlState.STOPPING:
		
		IF i_bStaAllStopped THEN
			s_eCtrlState := E_CtrlState.STOPPED;
		END_IF
		
ELSE
	s_eCtrlState := E_CtrlState.STOPPED;
END_CASE

IF (s_eCtrlState = E_CtrlState.STOPPED) THEN
	s_fbHmiBtnModeAutomatic.p_bStaEnabled := s_eCtrlMode <> E_CtrlMode.AUTOMATIC;
	s_fbHmiBtnModeManual.p_bStaEnabled := s_eCtrlMode <> E_CtrlMode.MANUAL;
	s_fbHmiBtnModeMaintenance.p_bStaEnabled := s_eCtrlMode <> E_CtrlMode.MAINTENANCE;
	s_fbHmiBtnModeIO.p_bStaEnabled := s_eCtrlMode <> E_CtrlMode.IO;
	s_fbHmiBtnModeCleaning.p_bStaEnabled := s_eCtrlMode <> E_CtrlMode.CLEANING;
ELSE
	s_fbHmiBtnModeAutomatic.p_bStaEnabled := FALSE;
	s_fbHmiBtnModeManual.p_bStaEnabled := FALSE;
	s_fbHmiBtnModeMaintenance.p_bStaEnabled := FALSE;
	s_fbHmiBtnModeIO.p_bStaEnabled := FALSE;
	s_fbHmiBtnModeCleaning.p_bStaEnabled := FALSE;
END_IF

IF (s_eCtrlMode <> E_CtrlMode.IDLE) THEN
	s_fbHmiBtnStateStart.p_bStaEnabled := s_eCtrlState = E_CtrlState.IDLE;
	s_fbHmiBtnStateStop.p_bStaEnabled := s_eCtrlState = E_CtrlState.RUNNING OR s_eCtrlState = E_CtrlState.IDLE;
	s_fbHmiBtnStateReset.p_bStaEnabled := s_eCtrlState = E_CtrlState.STOPPED;
ELSE
	s_fbHmiBtnStateStart.p_bStaEnabled := FALSE;
	s_fbHmiBtnStateStop.p_bStaEnabled := FALSE;
	s_fbHmiBtnStateReset.p_bStaEnabled := FALSE;
END_IF

_m_Devices := TRUE;
END_METHOD

METHOD PROTECTED _m_Init : BOOL

//Mode buttons
s_fbHmiBtnModeAutomatic.p_eButtontype := E_HmiButtonType.PUSHBUTTON;
s_fbHmiBtnModeAutomatic.p_bStaVisible := FALSE;
s_fbHmiBtnModeAutomatic.p_bStaEnabled := FALSE;
s_fbHmiBtnModeAutomatic.p_sBtnText := 'Automatic';

s_fbHmiBtnModeManual.p_eButtontype := E_HmiButtonType.PUSHBUTTON;
s_fbHmiBtnModeManual.p_bStaVisible := FALSE;
s_fbHmiBtnModeManual.p_bStaEnabled := FALSE;
s_fbHmiBtnModeManual.p_sBtnText := 'Manual';

s_fbHmiBtnModeMaintenance.p_eButtontype := E_HmiButtonType.PUSHBUTTON;
s_fbHmiBtnModeMaintenance.p_bStaVisible := FALSE;
s_fbHmiBtnModeMaintenance.p_bStaEnabled := FALSE;
s_fbHmiBtnModeMaintenance.p_sBtnText := 'Maintenance';

s_fbHmiBtnModeIO.p_eButtontype := E_HmiButtonType.PUSHBUTTON;
s_fbHmiBtnModeIO.p_bStaVisible := FALSE;
s_fbHmiBtnModeIO.p_bStaEnabled := FALSE;
s_fbHmiBtnModeIO.p_sBtnText := 'IO';

s_fbHmiBtnModeCleaning.p_eButtontype := E_HmiButtonType.PUSHBUTTON;
s_fbHmiBtnModeCleaning.p_bStaVisible := FALSE;
s_fbHmiBtnModeCleaning.p_bStaEnabled := FALSE;
s_fbHmiBtnModeCleaning.p_sBtnText := 'Cleaning';

//State buttons
s_fbHmiBtnStateStart.p_eButtontype := E_HmiButtonType.PUSHBUTTON;
s_fbHmiBtnStateStart.p_bStaVisible := FALSE;
s_fbHmiBtnStateStart.p_bStaEnabled := FALSE;
s_fbHmiBtnStateStart.p_sBtnText := 'Start';

s_fbHmiBtnStateStop.p_eButtontype := E_HmiButtonType.PUSHBUTTON;
s_fbHmiBtnStateStop.p_bStaVisible := FALSE;
s_fbHmiBtnStateStop.p_bStaEnabled := FALSE;
s_fbHmiBtnStateStop.p_sBtnText := 'Stop';

s_fbHmiBtnStateReset.p_eButtontype := E_HmiButtonType.PUSHBUTTON;
s_fbHmiBtnStateReset.p_bStaVisible := FALSE;
s_fbHmiBtnStateReset.p_bStaEnabled := FALSE;
s_fbHmiBtnStateReset.p_sBtnText := 'Reset';

_m_Init := TRUE;
END_METHOD

METHOD PUBLIC m_Main : BOOL

IF NOT s_bInitDone THEN
	IF _m_Init() THEN 
		s_bInitDone := TRUE;
	END_IF
END_IF

_m_Devices();

m_Main := TRUE;
END_METHOD

PROPERTY PUBLIC p_eCtrlMode : E_CtrlMode
GET

p_eCtrlMode := s_eCtrlMode;
END_GET
END_PROPERTY

PROPERTY PUBLIC p_eCtrlState : E_CtrlState
GET

p_eCtrlState := s_eCtrlState;
END_GET
END_PROPERTY

END_FUNCTION_BLOCK

// ---- POUs/General/FB_Flash.TcPOU
FUNCTION_BLOCK FB_Flash
VAR_INPUT
	i_bExcecute : BOOL;
	t_tOnTime : TIME := T#500MS;
	t_tOffTime : TIME := T#1S;;
END_VAR
VAR_OUTPUT
	o_bQ : BOOL;
END_VAR
VAR
	tonOn : TON;
	tonOff : TON;
	
END_VAR


tonOn(
	IN := i_bExcecute AND NOT(tonOff.Q),
	PT := t_tOnTime);
	
tonOff(
	IN := tonOn.Q,
	PT := t_tOffTime);
	
o_bQ := i_bExcecute AND NOT(tonOn.Q);

END_FUNCTION_BLOCK

// ---- POUs/General/FB_ForceOutput.TcPOU
FUNCTION_BLOCK FB_ForceOutput
VAR_INPUT
	i_ref_bCmdInput : REFERENCE TO BOOL;
	i_ref_bCmdOutput : REFERENCE TO BOOL;
	i_eForceValue : E_ForceValue := E_ForceValue.RELEASED;
END_VAR


IF i_eForceValue = E_ForceValue.RELEASED THEN
	i_ref_bCmdOutput := i_ref_bCmdInput;
ELSE
	i_ref_bCmdOutput := (i_eForceValue = E_ForceValue.FORCE_ON);
END_IF

END_FUNCTION_BLOCK

// ---- POUs/General/FB_InterlockHandler.TcPOU
FUNCTION_BLOCK FB_InterlockHandler
VAR_INPUT
	i_stInterlockList : ST_InterlockList;
END_VAR
VAR
	s_bInterlocked : BOOL;
	s_sReason : STRING(GVL.g_nMAX_LEN_REASON);
	i : USINT;
	s_nInterlockCnt : USINT;
	
END_VAR


s_bInterlocked := FALSE;
s_sReason := '';
s_nInterlockCnt := 0;

FOR i := 0 TO (GVL.g_nLEN_INTERLOCK_LIST-1) DO
	IF i_stInterlockList.arr_Interlocks[i].bState THEN
		s_bInterlocked := i_stInterlockList.arr_Interlocks[i].bState;
		s_sReason := i_stInterlockList.arr_Interlocks[i].sReason;
		EXIT;
	END_IF
END_FOR

PROPERTY PUBLIC p_bInterlocked : BOOL
GET

p_bInterlocked := s_bInterlocked;
END_GET
END_PROPERTY

PROPERTY PUBLIC p_sReason : STRING
GET

p_sReason := s_sReason;
END_GET
END_PROPERTY

PROPERTY PUBLIC p_stInterlock : ST_Interlock
GET

p_stInterlock.bState := s_bInterlocked;
p_stInterlock.sReason := s_sReason;
END_GET
END_PROPERTY

END_FUNCTION_BLOCK

// ---- POUs/General/FB_MovAvg.TcPOU
//This function calculates the moving avarage
//Based on the fuction below. 
//avg(n) = ( avg(n-1) * (n-1) + value(n) ) / n
FUNCTION_BLOCK FB_MovAvg
VAR_INPUT
	i_rIn : LREAL;
	i_nSamples : UINT;
END_VAR
VAR_OUTPUT
	o_rOut : LREAL;
END_VAR
VAR
	s_nSampleCounter : UINT := 0;
	s_rAvgPrev : LREAL := 0;
END_VAR


IF (s_nSampleCounter < i_nSamples) THEN
	s_nSampleCounter := s_nSampleCounter + 1;
END_IF

//Limit
IF s_nSampleCounter < 1 THEN
	s_nSampleCounter := 1;
ELSIF i_nSamples > 0 AND i_nSamples < s_nSampleCounter THEN
	s_nSampleCounter := i_nSamples;
END_IF

IF s_nSampleCounter = 1 THEN
	s_rAvgPrev := i_rIn;
END_IF

s_rAvgPrev := (s_rAvgPrev * (s_nSampleCounter-1) + i_rIn) / s_nSampleCounter;

o_rOut := s_rAvgPrev;

END_FUNCTION_BLOCK

// ---- POUs/General/FB_Toggle.TcPOU
FUNCTION_BLOCK FB_Toggle
VAR_INPUT
	CLK : BOOL;
END_VAR
VAR_OUTPUT
	Q : BOOL;
	osrQ : BOOL;
END_VAR
VAR
	s_osr : R_TRIG;
	s_osrQ : R_TRIG;
END_VAR


s_osr(CLK := CLK);

IF s_osr.Q AND Q THEN
	Q := FALSE; 
ELSIF s_osr.Q AND NOT(Q) THEN
	Q := TRUE;
END_IF

s_osrQ(CLK := Q);
osrQ := s_osrQ.Q;

END_FUNCTION_BLOCK

// ---- POUs/General/F_InRange.TcPOU
FUNCTION F_InRange : BOOL
VAR_INPUT
	i_fTargetValue : LREAL;
	i_fActualValue : LREAL;
	i_fRange : LREAL;
END_VAR
VAR
	s_fRange : LREAL;
END_VAR


IF i_fRange <= 0.0 THEN
	s_fRange := 0.1;
ELSE
	s_fRange := i_fRange;
END_IF

F_InRange := ( ABS(i_fTargetValue -  i_fActualValue) <= s_fRange );

END_FUNCTION

// ---- GlobalTextList.TcGTLO
TEXTLIST GlobalTextList
  292 = '   Q      State     Error'
  1145 = '#s'
  593 = '%'
  744 = '%s'
  670 = 'Actual mode:'
  459 = 'Actual step Centering:'
  734 = 'Actual step Transport:'
  384 = 'Actual step:'
  659 = 'Actual step: %c'
  904 = 'Actual step: %s'
  858 = 'Air'
  1193 = 'Air pressure OK'
  961 = 'ALARM LIST'
  567 = 'Apply'
  838 = 'Automatic'
  503 = 'Backward'
  60 = 'Brake'
  947 = 'Brake Released'
  315 = 'Button 1'
  574 = 'Button 2'
  341 = 'BWD'
  784 = 'CCW'
  856 = 'Center'
  642 = 'Centering'
  857 = 'Centering position'
  67 = 'Centering TB'
  698 = 'Clamps lower closed'
  469 = 'Clamps lower opened'
  800 = 'Clamps upper closed'
  639 = 'Clamps upper opened'
  668 = 'Close'
  268 = 'Close Inner Door'
  269 = 'CM Docking Clamp Lower'
  647 = 'CM Docking Clamp Upper'
  14 = 'CM Door Opener'
  1012 = 'CM Door Shutter'
  117 = 'CM Pallet Centering'
  1154 = 'CM Pallet Conveyor'
  240 = 'CM Unlocking Pin Lower'
  71 = 'CM Unlocking Pin Upper'
  314 = 'Cmd     State     Error'
  271 = 'CW'
  736 = 'Dock TB'
  843 = 'Docking'
  379 = 'Docking Clamp Lower'
  767 = 'Docking Clamp Upper'
  316 = 'Docking Interface'
  621 = 'Docking position'
  866 = 'Docking Station'
  715 = 'Docking System'
  1135 = 'Door'
  638 = 'Door opened'
  281 = 'Door Opener'
  157 = 'Door Shutter'
  113 = 'Drive Error'
  342 = 'Drive Running'
  1278 = 'EM Docking Interface'
  299 = 'EM Pallet Centering'
  359 = 'EM Pallet Conveyor'
  364 = 'Err'
  979 = 'Erro'
  381 = 'Error'
  338 = 'Export'
  1069 = 'Export Param'
  98 = 'Forward'
  324 = 'Front'
  782 = 'FWD'
  958 = 'High pressure'
  187 = 'Idle'
  1196 = 'Import'
  1324 = 'Import Param'
  439 = 'Infeed'
  114 = 'Infeed front'
  883 = 'Infeed front position'
  893 = 'Infeed rear'
  799 = 'Infeed rear position'
  376 = 'Left     Error'
  234 = 'Left     Right     Error'
  375 = 'Lock'
  192 = 'Main'
  848 = 'MainScreen'
  196 = 'Manual'
  445 = 'Motor'
  927 = 'Motor Stopped'
  675 = 'Motore'
  308 = 'Open'
  43 = 'Open Inner Door'
  104 = 'Opener almost closed'
  633 = 'Opener closed'
  769 = 'Opener opened'
  101 = 'Outer door opened'
  186 = 'Outer doorTB'
  674 = 'Outer TB'
  643 = 'Pallet Centering'
  933 = 'Pallet Conveyor'
  73 = 'Pallet Dectection'
  628 = 'Pallet Detection'
  254 = 'Pin lower locked'
  721 = 'Pin lower released'
  9 = 'Pin upper locked'
  677 = 'Pin upper released'
  693 = 'Power'
  115 = 'Power OK'
  276 = 'Q'
  387 = 'Q start/res'
  374 = 'Q start/reset'
  272 = 'qCCW'
  1022 = 'qCW'
  583 = 'qEnable'
  884 = 'Qrel'
  355 = 'Qrelay'
  172 = 'qRelay'
  49 = 'Qrelease'
  837 = 'Qreset'
  1180 = 'qReset'
  666 = 'Qrev'
  1008 = 'Qstart/reset'
  18 = 'Raw speed (Ai): %i'
  56 = 'Raw target speed (Ai): %i'
  796 = 'Raw target speed: %2.5f'
  812 = 'Raw target speed: %d4'
  270 = 'Raw target speed: %f1.1 mm/s'
  532 = 'Raw target speed: %f2 mm/s'
  112 = 'Raw target speed: %f3.1 mm/s'
  80 = 'Raw target speed: %i'
  623 = 'Raw target speed: %i mm/s'
  683 = 'Raw target speed: %i5'
  860 = 'Rear'
  952 = 'Release'
  783 = 'Released'
  258 = 'Reset'
  163 = 'Rest'
  888 = 'Reverse'
  813 = 'Run/Reset'
  1151 = 'Running'
  512 = 'Safety'
  697 = 'Safety OK'
  385 = 'sdf'
  703 = 'Shutter closed'
  510 = 'Shutter opened'
  944 = 'Speed'
  862 = 'Start / Reset'
  498 = 'State'
  322 = 'State     Error'
  616 = 'Stop'
  197 = 'Stopped'
  820 = 'Target speed: %i mm/s'
  393 = 'Target: %i mm/s'
  103 = 'TB to center'
  363 = 'TB to docking'
  537 = 'TB to Infeed'
  929 = 'Undock TB'
  1201 = 'Unlocking Pin Lower'
  474 = 'Unlocking Pin Upper'
  478 = 'Unlocking Pins Lower'
  255 = 'Unlocking Pins Upper'
  1088 = 'Utilities'
  896 = 'valve Error'
  1146 = 'Warning'
END_TEXTLIST
